// TIA Portal V17 export
// export: Created 2023-04-04T13:27:26.2250054Z, ExportSetting WithDefaults, DisplayName Totally Integrated Automation Portal, DisplayVersion V17, DisplayName TIA Portal Openness, DisplayVersion V17, DisplayName TIA Portal Version Control Interface, DisplayVersion V17, DisplayName STEP 7 Professional, DisplayVersion V17, DisplayName STEP 7 Safety, DisplayVersion V17, DisplayName WinCC Advanced, DisplayVersion V17
DATA_BLOCK "gtyp_Setup"   // DB23
TITLE = Global DB Setup
{ S7_Optimized_Access := 'TRUE' }
AUTHOR : A.Schaefer
VERSION : 0.0
// stored: AutoNumber true, DBAccessibleFromOPCUA true, DBAccessibleFromWebserver true, InstanceOfName typ_Setup, InstanceOfType UDT, IsOnlyStoredInLoadMemory false, IsWriteProtectedInAS false
"typ_Setup"
   // VAR
   //    r_Version_SPS : Real;
   //    x_Fill_Rack_HBW : Bool;
   //    x_Start_TON_Fill_HBW : Bool;
   //    x_Clean_Rack_HBW : Bool;
   //    x_Park_Position : Bool;
   //    x_AcknowledgeButton : Bool;
   //    x_Color_Sensor_Calibration : Bool;
   //    x_Set_Calib_Value_Color_Blue : Bool;
   //    x_Set_Calib_Value_Color_White : Bool;
   //    x_Set_Calib_Value_Color_Red : Bool;
   //    x_Calculate_Value_Color : Bool;
   //    i_Color_Sensor_Selection : Int;
   //    w_Calib_ColorValue_Blue : Word;
   //    w_Calib_ColorValue_White : Word;
   //    w_Calib_ColorValue_Red : Word;
   //    w_Threshold_White_Red : Word;
   //    w_Threshold_Red_Blue : Word;
   //    w_Actual_ColorValue : Word;
   //    x_Set_Pos_Activ : Bool;
   //    x_Start_Positioning : Bool;
   //    x_Final_Positioning : Bool;
   //    x_Home_Positioning : Bool;
   //    x_Start_Offset : Bool;
   //    i_Pos_Selection : Int;
   //    di_Pos_Horizontal : DInt;
   //    di_Pos_Vertical : DInt;
   //    di_Pos_Rotate : DInt;
   //    x_Counter_Value_Calibration : Bool;
   //    i_Calib_CounterValue_Blue : Int;
   //    i_Calib_CounterValue_White : Int;
   //    i_Calib_CounterValue_Red : Int;
   //    x_Set_CounterValues : Bool;
   //    x_Activate_Continuous_Operation : Bool;
   // END_VAR
BEGIN
END_DATA_BLOCK
